{attribute 'qualified_only'}
{attribute 'strict'}
TYPE E_Xbox_XPlanar_JogMode :
(
	Slow			:= 0,
	FastWithButton 	:= 1,
	FastWithTrigger := 2
);
END_TYPE

(* stored: Version 1.1.0.1, ProductVersion 3.1.4024.11
   DUT E_Xbox_XPlanar_JogMode: Id {e445b7b9-ea0c-031f-24d3-3a0485f57791} *)
